// TIA Portal V18 export
DATA_BLOCK "DB_AQ"   // DB9
{ S7_Optimized_Access := 'FALSE' }
VERSION : 0.1
// stored: AutoNumber true, DBAccessibleFromOPCUA true, DBAccessibleFromWebserver true, IsOnlyStoredInLoadMemory false, IsWriteProtectedInAS false
   VAR
      outa_BaseAxis : Real;
      outa_Arm1Axis : Real;
      outa_Arm2Axis : Real;
      outa_Arm3Axis : Real;
      outa_ToolAxis : Real;
      outa_BaseSpeed : Real;
      outa_Arm1Speed : Real;
      outa_Arm2Speed : Real;
      outa_Arm3Speed : Real;
      outa_ToolSpeed : Real;
      outa_10 : Real;
      outa_11 : Real;
      outa_HorizontalAxis : Real;
      outa_VerticalAxis : Real;
   END_VAR
BEGIN
END_DATA_BLOCK
